TYPE ST_CameraGridSettings :
STRUCT
  bValid            : BOOL;   // ?
  eCameraMode       : E_CameraMode;
  eDeformationType  : E_DeformationType;  // selected deformation type based on selecte camera and settings
  fGridFeaturePitch : LREAL;  // feature grid picth (cam frame width) [px]
  fDetectToCam      : LREAL;  // distance between detection and camera [m]
END_STRUCT
END_TYPE

(* stored: Version 1.1.0.1, ProductVersion 3.1.4024.11
   DUT ST_CameraGridSettings: Id {293e8458-b723-4738-9579-a918fe2ed0a7} *)
